// TIA Portal project "rmcs_V13_SP1_V14" (V14)

(* hardware
DEVICE "S7-1200 station_1"  SIMATIC 1200-Station
   slot 0: "S7-1200 rack"  Rack  V1.0
   slot 1: "PLC_1"  CPU 1214C DC/DC/DC  6ES7 214-1AG31-0XB0  V3.0
*)

// ===== PLC "PLC_1"  CPU 1214C DC/DC/DC =====

VAR_GLOBAL   // PLC tag table "Default tag table"
   "A+" AT %Q0.0 : Bool;
   "A-" AT %Q0.1 : Bool;
   "B+" AT %Q0.2 : Bool;
   "B-" AT %Q0.3 : Bool;
   "systemStart" AT %M0.0 : Bool;
   "swap" AT %M0.1 : Bool;
   "motor1" AT %Q1.0 : Bool;
END_VAR

DATA_BLOCK "data"   // DB1
{ S7_Optimized_Access := 'TRUE' }
VERSION : 0.1
   VAR
      system : Bool;
      motor : Bool;
      speed : Int;
      rotation : Int;
      temperature : Int := 0;
   END_VAR
BEGIN
END_DATA_BLOCK

// folder: System blocks/Program resources

DATA_BLOCK "IEC_Timer_0_DB_1"   // DB3
{ S7_Optimized_Access := 'TRUE' }
AUTHOR : Simatic
FAMILY : IEC
NAME : IEC_TMR
VERSION : 1.0
// stored: InstanceOfName IEC_TIMER
"IEC_TIMER"
BEGIN
END_DATA_BLOCK

DATA_BLOCK "IEC_Timer_0_DB_2"   // DB4
{ S7_Optimized_Access := 'TRUE' }
AUTHOR : Simatic
FAMILY : IEC
NAME : IEC_TMR
VERSION : 1.0
// stored: InstanceOfName IEC_TIMER
"IEC_TIMER"
BEGIN
END_DATA_BLOCK

DATA_BLOCK "IEC_Timer_0_DB_4"   // DB6
{ S7_Optimized_Access := 'TRUE' }
AUTHOR : Simatic
FAMILY : IEC
NAME : IEC_TMR
VERSION : 1.0
// stored: InstanceOfName IEC_TIMER
"IEC_TIMER"
BEGIN
END_DATA_BLOCK

DATA_BLOCK "IEC_Timer_0_DB_5"   // DB7
{ S7_Optimized_Access := 'TRUE' }
AUTHOR : Simatic
FAMILY : IEC
NAME : IEC_TMR
VERSION : 1.0
// stored: InstanceOfName IEC_TIMER
"IEC_TIMER"
BEGIN
END_DATA_BLOCK

// folder: (top level)

ORGANIZATION_BLOCK "Main"   // OB1, LAD, ProgramCycle
TITLE = "Main Program Sweep (Cycle)"
{ S7_Optimized_Access := 'TRUE' }
VERSION : 0.1
   VAR_TEMP
      RET_VAL : Int;
      TimerRet1 : Time;
      TimerRet2 : Time;
      TimerRet3 : Time;
      TimerRet4 : Time;
      TimerRet5 : Time;
      TimerRet6 : Time;
      DelayTime : DWord;
   END_VAR
BEGIN

REGION Network 1
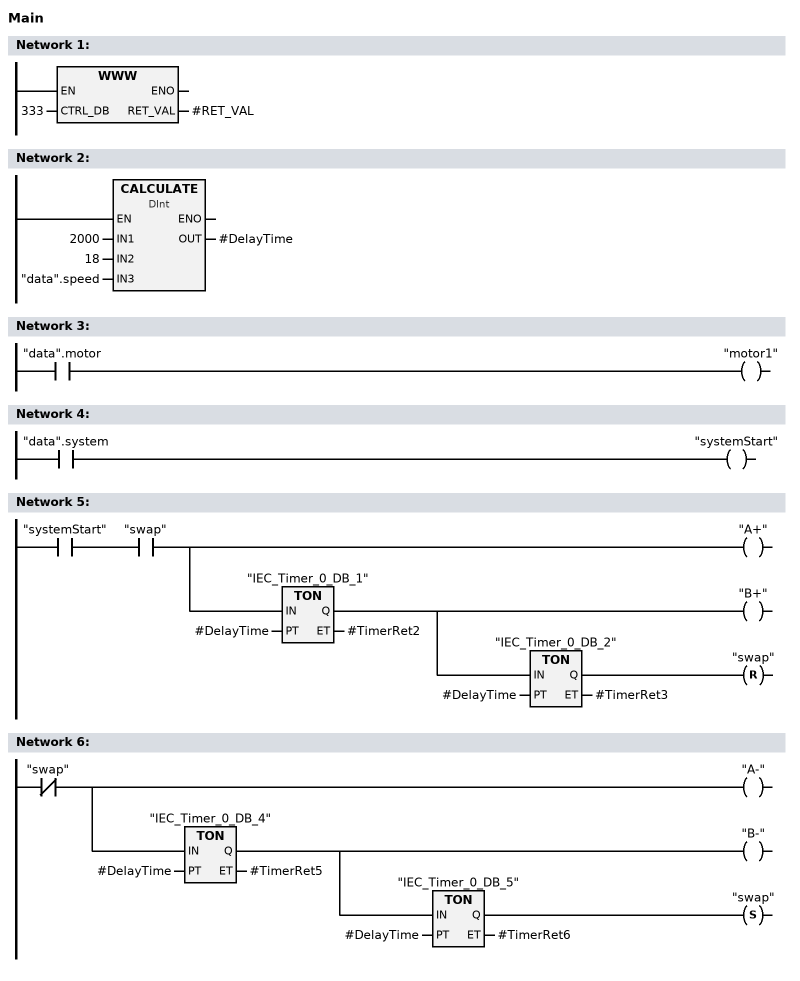
   #RET_VAL := WWW(CTRL_DB := 333);
END_REGION

REGION Network 2
   RUNG wire#powerrail
      { S7_Templates := "SrcType := DInt"; S7_GenerateENO := "TRUE"; S7_Expression := "IN1 - (IN2 * IN3)" } Calculate(in1 := 2000, in2 := 18, in3 := "data".speed, out => #DelayTime)
   END_RUNG
   // the same network as SCL:
   #DelayTime := 2000 - (18 * "data".speed);
END_REGION

REGION Network 3
   RUNG wire#powerrail
      Contact( "data".motor )
      Coil( "motor1" )
   END_RUNG
   // the same network as SCL:
   "motor1" := "data".motor;
END_REGION

REGION Network 4
   RUNG wire#powerrail
      Contact( "data".system )
      Coil( "systemStart" )
   END_RUNG
   // the same network as SCL:
   "systemStart" := "data".system;
END_REGION

REGION Network 5
   "A+" := "systemStart" AND "swap";
   "IEC_Timer_0_DB_1".TON(IN := "A+", PT := #DelayTime, ET => #TimerRet2);
   "B+" := "IEC_Timer_0_DB_1".Q;
   "IEC_Timer_0_DB_2".TON(IN := "IEC_Timer_0_DB_1".Q, PT := #DelayTime, ET => #TimerRet3);
   IF "IEC_Timer_0_DB_2".Q THEN "swap" := FALSE; END_IF;
END_REGION

REGION Network 6
   "A-" := NOT "swap";
   "IEC_Timer_0_DB_4".TON(IN := NOT "swap", PT := #DelayTime, ET => #TimerRet5);
   "B-" := "IEC_Timer_0_DB_4".Q;
   "IEC_Timer_0_DB_5".TON(IN := "IEC_Timer_0_DB_4".Q, PT := #DelayTime, ET => #TimerRet6);
   IF "IEC_Timer_0_DB_5".Q THEN "swap" := TRUE; END_IF;
END_REGION
END_ORGANIZATION_BLOCK